FUNCTION_BLOCK FB_InitialPos
VAR_INPUT
	bEnable : BOOL;
	fCurrentPos : LREAL;
END_VAR
VAR_OUTPUT
	fInitialPos : LREAL;
END_VAR
VAR
END_VAR

IF bEnable THEN
	fInitialPos := fInitialPos;
ELSE 
	fInitialPos := fCurrentPos;
END_IF

END_FUNCTION_BLOCK

(* stored: Version 1.1.0.1, ProductVersion 3.1.4024.12
   POU FB_InitialPos: Id {4f6abf03-5486-4a2c-ab9b-8b48fab2886b}, SpecialFunc None *)
